{attribute 'GeneratedUsingTerminal: EK1100-0000-0018'}
{attribute addProperty BoxType "EK1100-0000-0018"}
{attribute addProperty Id "Beckhoff_ER6xxxEK1122Beckhoff_ER6xxxEK1122_BD5112F1446"}
{attribute addProperty CRC "2305653150"}
{attribute addProperty Size "446"}
TYPE Beckhoff_ER6xxx_896D799E EXTENDS EK1100_1FC0878B :
STRUCT
	{attribute addProperty Name "Beckhoff_ER6xxxEK1122"}
	{attribute addProperty PreviousPort "Beckhoff ER6xxx : B"}
	Beckhoff_ER6xxxEK1122 : Beckhoff_ER6xxxEK1122_BD5112F1;
END_STRUCT
END_TYPE

(* stored: Version 1.2.0.0, ProductVersion 3.1.4024.9
   DUT Beckhoff_ER6xxx_896D799E: Id {921f7943-e994-44f5-bd85-27297d378eab} *)
